KUKA KRL program: ho_com_02_ag01_g01.src, ho_com_02_ag01_g01.dat

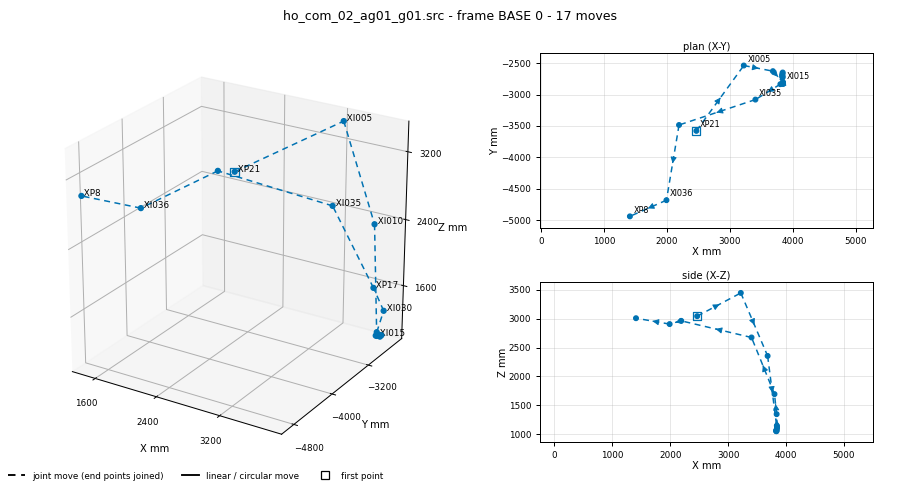
[picture p0: tool path of ho_com_02_ag01_g01.src in frame BASE 0, 17 of 17 moves have a stored position in this frame; points joined in program order, loops and branches not executed]
--- ho_com_02_ag01_g01.src ---
&ACCESS RVO4
&REL 568
&COMMENT Pega Traseira LTA-LTB
&PARAM DISKPATH = KRC:\R1\Program\MANIPULACAO NTC
DEF HO_COM_02_AG01_G01 ( )
;FOLD INI
  ;FOLD BASISTECH INI
    GLOBAL INTERRUPT DECL 3 WHEN $STOPMESS==TRUE DO IR_STOPM ( )
    INTERRUPT ON 3
    BAS (#INITMOV,0)
  ;ENDFOLD (BASISTECH INI)
;FOLD GRIPPERTECH INI
USER_GRP(0,DUMMY,DUMMY,GDEFAULT)
;ENDFOLD (GRIPPERTECH INI)
  ;FOLD USER INI
    ;Make your modifications here

  ;ENDFOLD (USER INI)
;ENDFOLD (INI)

; Caracterizacao dos meios de producao
; Changes: Pega Traseira no AGV
; Modelos: Axor/Atego - LTA/LTB
; Versao Atual: 05/01/2016
; Ferramenta: Gripper 903
; Name: P13.050-R1

chk_w9_wechs_ok ( ) ;CHECK GRIPPER 903

;FOLD PTP P21 CONT Vel=100 % PDAT15 Tool[10]:Grp 903 c/ pc Base[0];%{PE}%R 8.2.20,%MKUKATPBASIS,%CMOVE,%VPTP,%P 1:PTP, 2:P21, 3:C_DIS, 5:100, 7:PDAT15
$BWDSTART=FALSE
PDAT_ACT=PPDAT15
FDAT_ACT=FP21
BAS(#PTP_PARAMS,100)
PTP XP21 C_DIS
;ENDFOLD

;FOLD WAIT FOR ( NOT IN 581 'DK 8 GRP Axor 903 Tampa R' ) AND ( IN 582 'DK 8 GRP Axor 903 Tampa V' );%{PE}%R 8.2.20,%MKUKATPBASIS,%CEXT_WAIT_FOR,%VEXT_WAIT_FOR,%P 2:, 4:NOT, 5:$IN, 6:581, 7:DK 8 GRP Axor 903 Tampa R, 9:AND, 10:, 12:, 13:$IN, 14:582, 15:DK 8 GRP Axor 903 Tampa V, 17:
WAIT FOR  (  NOT $IN[581] ) AND ( $IN[582] )
;ENDFOLD
;FOLD WAIT FOR ( NOT IN 489 'Presença de peça 1 - Axor 903' ) AND ( NOT IN 490 'Presença de peça 2 - Axor 903' );%{PE}%R 8.2.20,%MKUKATPBASIS,%CEXT_WAIT_FOR,%VEXT_WAIT_FOR,%P 2:, 4:NOT, 5:$IN, 6:489, 7:Presença de peça 1 - Axor 903, 9:AND, 10:, 12:NOT, 13:$IN, 14:490, 15:Presença de peça 2 - Axor 903, 17:
WAIT FOR  (  NOT $IN[489] ) AND (  NOT $IN[490] )
;ENDFOLD

; ABRE GRAMPOS
;FOLD SET Z1.1/2 GRP AXOR 903 State=OPN CONT at START Delay=1 ms;%{PE}%R 8.2.1,%MKUKATPGRP,%CGRP,%VGRP,%P 2:7, 4:1, 5:#YES, 6:GDAT19, 8:0, 10:1
TRIGGER WHEN DISTANCE=0 DELAY=1 DO H50(GRP_APO,7,1,GCONT) PRIO=-1
;ENDFOLD
;FOLD SET Z2.1/2 RPS AXOR 903 State=OPN CONT at START Delay=1 ms;%{PE}%R 8.2.1,%MKUKATPGRP,%CGRP,%VGRP,%P 2:8, 4:1, 5:#YES, 6:GDAT23, 8:0, 10:1
TRIGGER WHEN DISTANCE=0 DELAY=1 DO H50(GRP_APO,8,1,GCONT) PRIO=-1
;ENDFOLD
;FOLD SET Z3.1 GRP AXOR 903 State=OPN CONT at START Delay=1 ms;%{PE}%R 8.2.1,%MKUKATPGRP,%CGRP,%VGRP,%P 2:9, 4:1, 5:#YES, 6:GDAT21, 8:0, 10:1
TRIGGER WHEN DISTANCE=0 DELAY=1 DO H50(GRP_APO,9,1,GCONT) PRIO=-1
;ENDFOLD
;FOLD SET Z7.1 GRP 7 AXOR 903 State=OPN CONT at START Delay=1 ms;%{PE}%R 8.2.1,%MKUKATPGRP,%CGRP,%VGRP,%P 2:14, 4:1, 5:#YES, 6:GDAT27, 8:0, 10:1
TRIGGER WHEN DISTANCE=0 DELAY=1 DO H50(GRP_APO,14,1,GCONT) PRIO=-1
;ENDFOLD
;FOLD SET Z6.1 VAC AXOR 903 State=CONT at START Delay=1 ms;%{PE}%R 8.2.1,%MKUKATPGRP,%CGRP,%VGRP,%P 2:13, 4:2, 5:#YES, 6:GDAT28, 8:0, 10:1
TRIGGER WHEN DISTANCE=0 DELAY=1 DO H50(GRP_APO,13,2,GCONT) PRIO=-1
;ENDFOLD
;FOLD SET Z6.1 VAC AXOR 903 State=OFF CONT at START Delay=1 ms;%{PE}%R 8.2.1,%MKUKATPGRP,%CGRP,%VGRP,%P 2:13, 4:3, 5:#YES, 6:GDAT29, 8:0, 10:1
TRIGGER WHEN DISTANCE=0 DELAY=1 DO H50(GRP_APO,13,3,GCONT) PRIO=-1
;ENDFOLD
chk_w9_grp1_opn( )
chk_w9_rps2_opn( )
chk_w9_grp3_opn( )
chk_w9_grp4_opn( )
chk_w9_grp5_vac_off( )

;AGUARDA LIBERACAO DE PEGA
;FOLD OUT 3370 'Lib. p/ Pegar Parede Traseira' State=TRUE ;%{PE}%R 8.2.20,%MKUKATPBASIS,%COUT,%VOUTX,%P 2:3370, 3:Lib. p/ Pegar Parede Traseira, 5:TRUE, 6:
$OUT[3370]=TRUE
;ENDFOLD
;FOLD WAIT FOR ( IN 3370 'Aguarda Lib. p/ Retirar Parede Traseira' );%{PE}%R 8.2.20,%MKUKATPBASIS,%CEXT_WAIT_FOR,%VEXT_WAIT_FOR,%P 2:, 4:, 5:$IN, 6:3370, 7:Aguarda Lib. p/ Retirar Parede Traseira, 9:
WAIT FOR  ( $IN[3370] )
;ENDFOLD
;FOLD OUT 3370 'Lib. p/ Pegar Parede Traseira' State=FALSE ;%{PE}%R 8.2.20,%MKUKATPBASIS,%COUT,%VOUTX,%P 2:3370, 3:Lib. p/ Pegar Parede Traseira, 5:FALSE, 6:
$OUT[3370]=FALSE
;ENDFOLD
;FOLD OUT 3342 'Fora area externa' State=FALSE ;%{PE}%R 8.2.20,%MKUKATPBASIS,%COUT,%VOUTX,%P 2:3342, 3:Fora area externa, 5:FALSE, 6:
$OUT[3342]=FALSE
;ENDFOLD

;FOLD PTP l005 CONT Vel=100 % P_OLP2 Tool[10]:Grp 903 c/ pc Base[0];%{PE}%R 8.2.20,%MKUKATPBASIS,%CMOVE,%VPTP,%P 1:PTP, 2:l005, 3:C_DIS, 5:100, 7:P_OLP2
$BWDSTART=FALSE
PDAT_ACT=PP_OLP2
FDAT_ACT=Fl005
BAS(#PTP_PARAMS,100)
PTP Xl005 C_DIS
;ENDFOLD
;FOLD PTP l010 CONT Vel=100 % P_OLP3 Tool[10]:Grp 903 c/ pc Base[0];%{PE}%R 8.2.20,%MKUKATPBASIS,%CMOVE,%VPTP,%P 1:PTP, 2:l010, 3:C_DIS, 5:100, 7:P_OLP3
$BWDSTART=FALSE
PDAT_ACT=PP_OLP3
FDAT_ACT=Fl010
BAS(#PTP_PARAMS,100)
PTP Xl010 C_DIS
;ENDFOLD
;FOLD PTP l015 CONT Vel=100 % P_OLP4 Tool[10]:Grp 903 c/ pc Base[0];%{PE}%R 8.2.20,%MKUKATPBASIS,%CMOVE,%VPTP,%P 1:PTP, 2:l015, 3:C_DIS, 5:100, 7:P_OLP4
$BWDSTART=FALSE
PDAT_ACT=PP_OLP4
FDAT_ACT=Fl015
BAS(#PTP_PARAMS,100)
PTP Xl015 C_DIS
;ENDFOLD
;FOLD LIN P15 CONT Vel=2 m/s CPDAT3 Tool[10]:Grp 903 c/ pc Base[0];%{PE}%R 8.2.20,%MKUKATPBASIS,%CMOVE,%VLIN,%P 1:LIN, 2:P15, 3:C_DIS C_DIS, 5:2, 7:CPDAT3
$BWDSTART=FALSE
LDAT_ACT=LCPDAT3
FDAT_ACT=FP15
BAS(#CP_PARAMS,2)
LIN XP15 C_DIS C_DIS
;ENDFOLD
;FOLD LIN P9 CONT Vel=1 m/s CPDAT1 Tool[10]:Grp 903 c/ pc Base[0];%{PE}%R 8.2.20,%MKUKATPBASIS,%CMOVE,%VLIN,%P 1:LIN, 2:P9, 3:C_DIS C_DIS, 5:1, 7:CPDAT1
$BWDSTART=FALSE
LDAT_ACT=LCPDAT1
FDAT_ACT=FP9
BAS(#CP_PARAMS,1)
LIN XP9 C_DIS C_DIS
;ENDFOLD

; POSICAO DE PEGA AXOR/ATEGO LTA-LTB
;FOLD LIN P_PE02 Vel=0.25 m/s CPDAT4 Tool[9]:Grp 903 s/ pc Base[0];%{PE}%R 8.2.20,%MKUKATPBASIS,%CMOVE,%VLIN,%P 1:LIN, 2:P_PE02, 3:, 5:0.25, 7:CPDAT4
$BWDSTART=FALSE
LDAT_ACT=LCPDAT4
FDAT_ACT=FP_PE02
BAS(#CP_PARAMS,0.25)
LIN XP_PE02
;ENDFOLD

IF (NOT(GHOST())) THEN
;FOLD WAIT FOR ( IN 489 'Presença de peça 1 - Axor 903' ) AND ( IN 490 'Presença de peça 2 - Axor 903' );%{PE}%R 8.2.20,%MKUKATPBASIS,%CEXT_WAIT_FOR,%VEXT_WAIT_FOR,%P 2:, 4:, 5:$IN, 6:489, 7:Presença de peça 1 - Axor 903, 9:AND, 10:, 12:, 13:$IN, 14:490, 15:Presença de peça 2 - Axor 903, 17:
WAIT FOR  ( $IN[489] ) AND ( $IN[490] )
;ENDFOLD
ENDIF

; FECHA GRAMPOS
;FOLD SET Z2.1/2 RPS AXOR 903 State=CLO GDAT22;%{PE}%R 8.2.1,%MKUKATPGRP,%CGRP,%VGRP,%P 2:8, 4:2, 5:#NO, 6:GDAT22, 8:0, 10:0
H50(GRP,8,2,GGDAT22)
;ENDFOLD
;FOLD SET Z1.1/2 GRP AXOR 903 State=CLO GDAT16;%{PE}%R 8.2.1,%MKUKATPGRP,%CGRP,%VGRP,%P 2:7, 4:2, 5:#NO, 6:GDAT16, 8:0, 10:0
H50(GRP,7,2,GGDAT16)
;ENDFOLD
;FOLD SET Z3.1 GRP AXOR 903 State=CLO GDAT18;%{PE}%R 8.2.1,%MKUKATPGRP,%CGRP,%VGRP,%P 2:9, 4:2, 5:#NO, 6:GDAT18, 8:0, 10:0
H50(GRP,9,2,GGDAT18)
;ENDFOLD
;FOLD SET Z7.1 GRP 7 AXOR 903 State=CLO GDAT32;%{PE}%R 8.2.1,%MKUKATPGRP,%CGRP,%VGRP,%P 2:14, 4:2, 5:#NO, 6:GDAT32, 8:0, 10:0
H50(GRP,14,2,GGDAT32)
;ENDFOLD
chk_w9_rps2_clo( )
chk_w9_grp1_clo( )
chk_w9_grp3_clo( )
chk_w9_grp4_clo( )

IF (NOT(GHOST())) THEN
;FOLD SET Z6.1 VAC AXOR 903 State=VACUUM GDAT31;%{PE}%R 8.2.1,%MKUKATPGRP,%CGRP,%VGRP,%P 2:13, 4:1, 5:#NO, 6:GDAT31, 8:0, 10:0
H50(GRP,13,1,GGDAT31)
;ENDFOLD
chk_w9_grp5_vac_on( )
ENDIF

;AGUARDA LIBERACAO SAIR COM PECA
;FOLD OUT 3371 'Lib. p/ Sair c/ Parede Traseira' State=TRUE ;%{PE}%R 8.2.20,%MKUKATPBASIS,%COUT,%VOUTX,%P 2:3371, 3:Lib. p/ Sair c/ Parede Traseira, 5:TRUE, 6:
$OUT[3371]=TRUE
;ENDFOLD
;FOLD WAIT FOR ( IN 3371 'Aguarda Lib. p/ Sair c/ Parede Traseira' );%{PE}%R 8.2.20,%MKUKATPBASIS,%CEXT_WAIT_FOR,%VEXT_WAIT_FOR,%P 2:, 4:, 5:$IN, 6:3371, 7:Aguarda Lib. p/ Sair c/ Parede Traseira, 9:
WAIT FOR  ( $IN[3371] )
;ENDFOLD
;FOLD OUT 3371 'Lib. p/ Sair c/ Parede Traseira' State=FALSE ;%{PE}%R 8.2.20,%MKUKATPBASIS,%COUT,%VOUTX,%P 2:3371, 3:Lib. p/ Sair c/ Parede Traseira, 5:FALSE, 6:
$OUT[3371]=FALSE
;ENDFOLD
;FOLD WAIT FOR ( IN 582 'DK 8 GRP Axor 903 Tampa V' );%{PE}%R 8.2.20,%MKUKATPBASIS,%CEXT_WAIT_FOR,%VEXT_WAIT_FOR,%P 2:, 4:, 5:$IN, 6:582, 7:DK 8 GRP Axor 903 Tampa V, 9:
WAIT FOR  ( $IN[582] )
;ENDFOLD

;FOLD LIN P11 Vel=0.25 m/s CPDAT2 Tool[10]:Grp 903 c/ pc Base[0];%{PE}%R 8.2.20,%MKUKATPBASIS,%CMOVE,%VLIN,%P 1:LIN, 2:P11, 3:, 5:0.25, 7:CPDAT2
$BWDSTART=FALSE
LDAT_ACT=LCPDAT2
FDAT_ACT=FP11
BAS(#CP_PARAMS,0.25)
LIN XP11
;ENDFOLD

IF (NOT(GHOST())) THEN
;FOLD WAIT FOR ( IN 489 'Presença de peça 1 - Axor 903' ) AND ( IN 490 'Presença de peça 2 - Axor 903' );%{PE}%R 8.2.20,%MKUKATPBASIS,%CEXT_WAIT_FOR,%VEXT_WAIT_FOR,%P 2:, 4:, 5:$IN, 6:489, 7:Presença de peça 1 - Axor 903, 9:AND, 10:, 12:, 13:$IN, 14:490, 15:Presença de peça 2 - Axor 903, 17:
WAIT FOR  ( $IN[489] ) AND ( $IN[490] )
;ENDFOLD
ENDIF

;FOLD LIN l020 CONT Vel=0.4 m/s L_OLP2 Tool[10]:Grp 903 c/ pc Base[0];%{PE}%R 8.2.20,%MKUKATPBASIS,%CMOVE,%VLIN,%P 1:LIN, 2:l020, 3:C_DIS C_DIS, 5:0.4, 7:L_OLP2
$BWDSTART=FALSE
LDAT_ACT=LL_OLP2
FDAT_ACT=Fl020
BAS(#CP_PARAMS,0.4)
LIN Xl020 C_DIS C_DIS
;ENDFOLD
;FOLD PTP P10 CONT Vel=100 % PDAT5 Tool[10]:Grp 903 c/ pc Base[0];%{PE}%R 8.2.20,%MKUKATPBASIS,%CMOVE,%VPTP,%P 1:PTP, 2:P10, 3:C_DIS, 5:100, 7:PDAT5
$BWDSTART=FALSE
PDAT_ACT=PPDAT5
FDAT_ACT=FP10
BAS(#PTP_PARAMS,100)
PTP XP10 C_DIS
;ENDFOLD
;FOLD PTP P12 CONT Vel=100 % PDAT6 Tool[10]:Grp 903 c/ pc Base[0];%{PE}%R 8.2.20,%MKUKATPBASIS,%CMOVE,%VPTP,%P 1:PTP, 2:P12, 3:C_DIS, 5:100, 7:PDAT6
$BWDSTART=FALSE
PDAT_ACT=PPDAT6
FDAT_ACT=FP12
BAS(#PTP_PARAMS,100)
PTP XP12 C_DIS
;ENDFOLD
;FOLD PTP l030 CONT Vel=50 % P_OLP6 Tool[10]:Grp 903 c/ pc Base[0];%{PE}%R 8.2.20,%MKUKATPBASIS,%CMOVE,%VPTP,%P 1:PTP, 2:l030, 3:C_DIS, 5:50, 7:P_OLP6
$BWDSTART=FALSE
PDAT_ACT=PP_OLP6
FDAT_ACT=Fl030
BAS(#PTP_PARAMS,50)
PTP Xl030 C_DIS
;ENDFOLD
;FOLD PTP P17 CONT Vel=50 % PDAT10 Tool[10]:Grp 903 c/ pc Base[0];%{PE}%R 8.2.20,%MKUKATPBASIS,%CMOVE,%VPTP,%P 1:PTP, 2:P17, 3:C_DIS, 5:50, 7:PDAT10
$BWDSTART=FALSE
PDAT_ACT=PPDAT10
FDAT_ACT=FP17
BAS(#PTP_PARAMS,50)
PTP XP17 C_DIS
;ENDFOLD
;FOLD PTP l035 CONT Vel=50 % P_OLP7 Tool[10]:Grp 903 c/ pc Base[0];%{PE}%R 8.2.20,%MKUKATPBASIS,%CMOVE,%VPTP,%P 1:PTP, 2:l035, 3:C_DIS, 5:50, 7:P_OLP7
$BWDSTART=FALSE
PDAT_ACT=PP_OLP7
FDAT_ACT=Fl035
BAS(#PTP_PARAMS,50)
PTP Xl035 C_DIS
;ENDFOLD
;FOLD PTP P18 CONT Vel=30 % PDAT11 Tool[10]:Grp 903 c/ pc Base[0];%{PE}%R 8.2.20,%MKUKATPBASIS,%CMOVE,%VPTP,%P 1:PTP, 2:P18, 3:C_DIS, 5:30, 7:PDAT11
$BWDSTART=FALSE
PDAT_ACT=PPDAT11
FDAT_ACT=FP18
BAS(#PTP_PARAMS,30)
PTP XP18 C_DIS
;ENDFOLD
;FOLD PTP l036 CONT Vel=30 % P_OLP9 Tool[10]:Grp 903 c/ pc Base[0];%{PE}%R 8.2.20,%MKUKATPBASIS,%CMOVE,%VPTP,%P 1:PTP, 2:l036, 3:C_DIS, 5:30, 7:P_OLP9
$BWDSTART=FALSE
PDAT_ACT=PP_OLP9
FDAT_ACT=Fl036
BAS(#PTP_PARAMS,30)
PTP Xl036 C_DIS
;ENDFOLD

;LIBERA AREA
;FOLD PULSE 3349 'R1 pegou peça' State=TRUE Time=3 sec;%{PE}%R 8.2.20,%MKUKATPBASIS,%COUT,%VPULSE,%P 2:3349, 3:R1 pegou peça, 5:TRUE, 6:, 8:3
PULSE($OUT[3349], TRUE,3)
;ENDFOLD
;FOLD OUT 3342 'Fora area externa' State=TRUE ;%{PE}%R 8.2.20,%MKUKATPBASIS,%COUT,%VOUTX,%P 2:3342, 3:Fora area externa, 5:TRUE, 6:
$OUT[3342]=TRUE
;ENDFOLD

;FOLD PTP P8 CONT Vel=30 % PDAT4 Tool[10]:Grp 903 c/ pc Base[0];%{PE}%R 8.2.20,%MKUKATPBASIS,%CMOVE,%VPTP,%P 1:PTP, 2:P8, 3:C_DIS, 5:30, 7:PDAT4
$BWDSTART=FALSE
PDAT_ACT=PPDAT4
FDAT_ACT=FP8
BAS(#PTP_PARAMS,30)
PTP XP8 C_DIS
;ENDFOLD

END

--- ho_com_02_ag01_g01.dat ---
&ACCESS RVO4
&REL 568
&COMMENT Pega Traseira LTA-LTB
&PARAM DISKPATH = KRC:\R1\Program\MANIPULACAO NTC
DEFDAT  ho_com_02_ag01_g01
;FOLD EXTERNAL DECLARATIONS;%{PE}%MKUKATPBASIS,%CEXT,%VCOMMON,%P
;FOLD GRIPPERTECH EXT
EXT  H50 (INT  :IN,INT  :IN,INT  :IN,GRP_TYP  :IN )
;ENDFOLD (GRIPPERTECH EXT)
;FOLD SPOTTECH EXT
EXT  USERSPOT (S_COMMAND  :IN,SPOT_TYPE  :IN )
;ENDFOLD (SPOTTECH EXT)
;FOLD BASISTECH EXT;%{PE}%MKUKATPBASIS,%CEXT,%VEXT,%P
EXT  BAS (BAS_COMMAND  :IN,REAL  :IN )
DECL INT SUCCESS
;ENDFOLD (BASISTECH EXT)
;FOLD USER EXT;%{E}%MKUKATPUSER,%CEXT,%VEXT,%P
;Make your modifications here

;ENDFOLD (USER EXT)
DECL FDAT Fl005={TOOL_NO 9,BASE_NO 0,IPO_FRAME #BASE,POINT2[] " ",TQ_STATE FALSE}
DECL PDAT PP_OLP2={VEL 100.0,ACC 100.0,APO_DIST 10.0,APO_MODE #CDIS}
DECL E6POS Xl005={X 3218.60791,Y -2539.229,Z 3442.36011,A -30.2562904,B 46.8825684,C -113.404999,S 2,T 11,E1 -3250.0,E2 0.0,E3 0.0,E4 0.0,E5 0.0,E6 0.0}
DECL FDAT Fl010={TOOL_NO 9,BASE_NO 0,IPO_FRAME #BASE,POINT2[] " "}
DECL PDAT PP_OLP3={VEL 100.0,ACC 100.0,APO_DIST 10.0,APO_MODE #CDIS}
DECL E6POS Xl010={X 3681.40308,Y -2628.80493,Z 2354.81299,A -52.0649681,B 58.5603714,C -139.654205,S 2,T 11,E1 -3426.1709,E2 0.0,E3 0.0,E4 0.0,E5 0.0,E6 0.0}
DECL FDAT Fl015={TOOL_NO 9,BASE_NO 0,IPO_FRAME #BASE,POINT2[] " "}
DECL PDAT PP_OLP4={VEL 100.0,ACC 100.0,APO_DIST 10.0,APO_MODE #CDIS}
DECL E6POS Xl015={X 3842.71606,Y -2807.72095,Z 1105.85901,A -89.6218338,B 67.1568527,C 178.501907,S 2,T 11,E1 -3522.73389,E2 0.0,E3 0.0,E4 0.0,E5 0.0,E6 0.0}
DECL FDAT FP_PE02={TOOL_NO 9,BASE_NO 0,IPO_FRAME #BASE,POINT2[] " ",TQ_STATE FALSE}
DECL E6POS XP_PE02={X 3830.49609,Y -2675.78906,Z 1055.40906,A -88.9839935,B 65.9510117,C 179.429596,S 2,T 11,E1 -3701.05493,E2 0.0,E3 0.0,E4 0.0,E5 0.0,E6 0.0}
DECL FDAT Fl020={TOOL_NO 10,BASE_NO 0,IPO_FRAME #BASE,POINT2[] " "}
DECL E6POS Xl020={X 3835.47607,Y -2731.25488,Z 1079.94604,A -89.6218033,B 67.1567001,C 178.501999,S 2,T 11,E1 -3700.23511,E2 0.0,E3 0.0,E4 0.0,E5 0.0,E6 0.0}
DECL LDAT LL_OLP2={VEL 0.25,ACC 100.0,APO_DIST 30.0,APO_FAC 0.0,ORI_TYP #VAR,CIRC_TYP #BASE,JERK_FAC 50.0}
DECL FDAT Fl030={TOOL_NO 10,BASE_NO 0,IPO_FRAME #BASE,POINT2[] " "}
DECL PDAT PP_OLP6={VEL 100.0,ACC 70.0,APO_DIST 50.0,APO_MODE #CDIS}
DECL E6POS Xl030={X 3837.04712,Y -2650.14209,Z 1349.71301,A 0.0,B 89.9999466,C -92.2000885,S 2,T 11,E1 -3700.00098,E2 0.0,E3 0.0,E4 0.0,E5 0.0,E6 0.0}
DECL FDAT Fl035={TOOL_NO 10,BASE_NO 0,IPO_FRAME #BASE,POINT2[] " ",TQ_STATE FALSE}
DECL PDAT PP_OLP7={VEL 100.0,ACC 50.0,APO_DIST 50.0,APO_MODE #CDIS}
DECL E6POS Xl035={X 3403.61108,Y -3080.45508,Z 2673.61792,A 76.7603836,B 73.9680481,C -4.25617409,S 2,T 11,E1 -3973.10107,E2 0.0,E3 0.0,E4 0.0,E5 0.0,E6 0.0}
DECL BASIS_SUGG_T LAST_BASIS={POINT1[] "P22                     ",POINT2[] "P22                     ",CP_PARAMS[] "CPDAT3                  ",PTP_PARAMS[] "PDAT16                  ",CONT[] "                        ",CP_VEL[] "0.4                     ",PTP_VEL[] "100                     ",SYNC_PARAMS[] "SYNCDAT                 ",SPL_NAME[] "S0                      "}
DECL PDAT PP_OLP9={VEL 100.0,ACC 50.0,APO_DIST 50.0,APO_MODE #CDIS}
DECL E6POS Xl036={X 1989.90601,Y -4679.04883,Z 2904.58691,A -29.6459503,B 80.8687363,C -48.2684593,S 2,T 11,E1 -3220.72095,E2 0.0,E3 0.0,E4 0.0,E5 0.0,E6 0.0}
DECL FDAT Fl036={TOOL_NO 10,BASE_NO 0,IPO_FRAME #BASE,POINT2[] " ",TQ_STATE FALSE}
DECL GRP_SUGG_T LAST_GRP={NUMBER[] "13                      ",STATE[] "3                       ",PARAMS[] "GDAT29                  "}
DECL GRP_TYP GGDAT4={G_APO #NO,GRP_TIME 0.200000003,CTRL #OFF,DLY 0,DST 1}
DECL GRP_TYP GGDAT6={G_APO #NO,GRP_TIME 0.200000003,CTRL #OFF,DLY 0,DST 1}
DECL GRP_TYP GGDAT8={G_APO #NO,GRP_TIME 0.200000003,CTRL #OFF,DLY 0,DST 1}
DECL GRP_TYP GGDAT5={G_APO #NO,GRP_TIME 0.200000003,CTRL #OFF,DLY 0,DST 1}
DECL GRP_TYP GGDAT7={G_APO #NO,GRP_TIME 0.200000003,CTRL #OFF,DLY 0,DST 1}
DECL GRP_TYP GGDAT9={G_APO #NO,GRP_TIME 0.200000003,CTRL #OFF,DLY 0,DST 1}
DECL GRP_TYP GGDAT10={G_APO #NO,GRP_TIME 0.200000003,CTRL #OFF,DLY 0,DST 1}
DECL GRP_TYP GGDAT11={G_APO #NO,GRP_TIME 0.200000003,CTRL #OFF,DLY 0,DST 1}
DECL GRP_TYP GGDAT12={G_APO #NO,GRP_TIME 0.200000003,CTRL #OFF,DLY 0,DST 1}
DECL GRP_TYP GGDAT13={G_APO #NO,GRP_TIME 0.200000003,CTRL #OFF,DLY 0,DST 1}
DECL GRP_TYP GGDAT14={G_APO #NO,GRP_TIME 0.200000003,CTRL #OFF,DLY 0,DST 1}
DECL GRP_TYP GGDAT15={G_APO #NO,GRP_TIME 0.200000003,CTRL #OFF,DLY 0,DST 1}
DECL GRP_TYP GGDAT16={G_APO #NO,GRP_TIME 0.200000003,CTRL #OFF,DLY 0,DST 1}
DECL GRP_TYP GGDAT17={G_APO #NO,GRP_TIME 0.200000003,CTRL #OFF,DLY 0,DST 1}
DECL GRP_TYP GGDAT18={G_APO #NO,GRP_TIME 0.200000003,CTRL #OFF,DLY 0,DST 1}
DECL E6POS XP8={X 1408.87598,Y -4935.90723,Z 3006.11108,A -20.0040207,B 69.0891495,C -21.5691395,S 2,T 11,E1 -3220.81396,E2 0.0,E3 0.0,E4 0.0,E5 0.0,E6 0.0}
DECL FDAT FP8={TOOL_NO 10,BASE_NO 0,IPO_FRAME #BASE,POINT2[] " ",TQ_STATE FALSE}
DECL PDAT PPDAT4={VEL 100.0,ACC 50.0,APO_DIST 50.0,APO_MODE #CDIS}
DECL GRP_TYP GGDAT19={G_APO #NO,GRP_TIME 0.200000003,CTRL #OFF,DLY 0,DST 1}
DECL GRP_TYP GGDAT20={G_APO #NO,GRP_TIME 0.200000003,CTRL #OFF,DLY 0,DST 1}
DECL GRP_TYP GGDAT21={G_APO #NO,GRP_TIME 0.200000003,CTRL #OFF,DLY 0,DST 1}
DECL E6POS XP9={X 3831.39795,Y -2694.11499,Z 1062.47095,A -89.3210831,B 67.2410583,C 178.401596,S 2,T 11,E1 -3706.729,E2 0.0,E3 0.0,E4 0.0,E5 0.0,E6 0.0}
DECL FDAT FP9={TOOL_NO 9,BASE_NO 0,IPO_FRAME #BASE,POINT2[] " ",TQ_STATE FALSE}
DECL LDAT LCPDAT1={VEL 2.0,ACC 100.0,APO_DIST 50.0,APO_FAC 50.0,AXIS_VEL 100.0,AXIS_ACC 100.0,ORI_TYP #VAR,CIRC_TYP #BASE,JERK_FAC 50.0,GEAR_JERK 50.0,EXAX_IGN 0}
DECL E6POS XP10={X 3843.63696,Y -2833.05688,Z 1120.75305,A -90.5353394,B 75.7654572,C 177.633301,S 2,T 11,E1 -3700.06592,E2 0.0,E3 0.0,E4 0.0,E5 0.0,E6 0.0}
DECL FDAT FP10={TOOL_NO 10,BASE_NO 0,IPO_FRAME #BASE,POINT2[] " ",TQ_STATE FALSE}
DECL PDAT PPDAT5={VEL 100.0,ACC 100.0,APO_DIST 30.0,APO_MODE #CDIS}
DECL E6POS XP11={X 3832.33203,Y -2715.6731,Z 1068.93896,A -89.3303986,B 65.348587,C 178.376099,S 2,T 11,E1 -3700.04199,E2 0.0,E3 0.0,E4 0.0,E5 0.0,E6 0.0}
DECL FDAT FP11={TOOL_NO 10,BASE_NO 0,IPO_FRAME #BASE,POINT2[] " ",TQ_STATE FALSE}
DECL LDAT LCPDAT2={VEL 2.0,ACC 100.0,APO_DIST 5.0,APO_FAC 50.0,AXIS_VEL 100.0,AXIS_ACC 100.0,ORI_TYP #VAR,CIRC_TYP #BASE,JERK_FAC 50.0,GEAR_JERK 50.0,EXAX_IGN 0}
DECL E6POS XP12={X 3840.92993,Y -2806.29492,Z 1150.78198,A -88.0371933,B 77.8013535,C -179.918396,S 2,T 11,E1 -3700.88989,E2 0.0,E3 0.0,E4 0.0,E5 0.0,E6 0.0}
DECL FDAT FP12={TOOL_NO 10,BASE_NO 0,IPO_FRAME #BASE,POINT2[] " ",TQ_STATE FALSE}
DECL PDAT PPDAT6={VEL 100.0,ACC 100.0,APO_DIST 30.0,APO_MODE #CDIS}
DECL LDAT LCPDAT3={VEL 2.0,ACC 100.0,APO_DIST 50.0,APO_FAC 50.0,AXIS_VEL 100.0,AXIS_ACC 100.0,ORI_TYP #VAR,CIRC_TYP #BASE,JERK_FAC 50.0,GEAR_JERK 50.0,EXAX_IGN 0}
DECL E6POS XP15={X 3833.42603,Y -2714.77393,Z 1055.72803,A -89.0524368,B 67.2397308,C 178.692993,S 2,T 11,E1 -3703.71997,E2 0.0,E3 0.0,E4 0.0,E5 0.0,E6 0.0}
DECL FDAT FP15={TOOL_NO 9,BASE_NO 0,IPO_FRAME #BASE,POINT2[] " ",TQ_STATE FALSE}
DECL GRP_TYP GGDAT22={G_APO #NO,GRP_TIME 0.200000003,CTRL #OFF,DLY 0,DST 1}
DECL GRP_TYP GGDAT23={G_APO #NO,GRP_TIME 0.200000003,CTRL #OFF,DLY 0,DST 1}
DECL GRP_TYP GGDAT3={G_APO #NO,GRP_TIME 0.200000003,CTRL #OFF,DLY 0,DST 1}
DECL GRP_TYP GGDAT1={G_APO #NO,GRP_TIME 0.200000003,CTRL #OFF,DLY 0,DST 1}
DECL GRP_TYP GGDAT2={G_APO #NO,GRP_TIME 0.200000003,CTRL #OFF,DLY 0,DST 1}
DECL GRP_TYP GGDAT24={G_APO #NO,GRP_TIME 0.200000003,CTRL #OFF,DLY 0,DST 1}
DECL E6POS XP17={X 3800.02808,Y -2835.55811,Z 1695.61401,A 77.3357925,B 87.3917465,C -11.0309896,S 2,T 11,E1 -3820.08398,E2 0.0,E3 0.0,E4 0.0,E5 0.0,E6 0.0}
DECL FDAT FP17={TOOL_NO 10,BASE_NO 0,IPO_FRAME #BASE,POINT2[] " ",TQ_STATE FALSE}
DECL PDAT PPDAT10={VEL 100.0,ACC 50.0,APO_DIST 50.0,APO_MODE #CDIS}
DECL E6POS XP18={X 2189.81909,Y -3484.28491,Z 2960.64111,A -23.6490192,B 79.1503906,C -53.971241,S 2,T 11,E1 -2223.51489,E2 0.0,E3 0.0,E4 0.0,E5 0.0,E6 0.0}
DECL FDAT FP18={TOOL_NO 10,BASE_NO 0,IPO_FRAME #BASE,POINT2[] " ",TQ_STATE FALSE}
DECL PDAT PPDAT11={VEL 100.0,ACC 50.0,APO_DIST 50.0,APO_MODE #CDIS}
DECL LDAT LCPDAT4={VEL 2.0,ACC 100.0,APO_DIST 100.0,APO_FAC 50.0,AXIS_VEL 100.0,AXIS_ACC 100.0,ORI_TYP #VAR,CIRC_TYP #BASE,JERK_FAC 50.0,GEAR_JERK 50.0,EXAX_IGN 0}
DECL GRP_TYP GGDAT25={G_APO #NO,GRP_TIME 0.200000003,CTRL #OFF,DLY 0,DST 1}
DECL GRP_TYP GGDAT26={G_APO #NO,GRP_TIME 0.200000003,CTRL #OFF,DLY 0,DST 1}
DECL GRP_TYP GGDAT27={G_APO #NO,GRP_TIME 0.200000003,CTRL #OFF,DLY 0,DST 1}
DECL GRP_TYP GGDAT28={G_APO #NO,GRP_TIME 0.200000003,CTRL #OFF,DLY 0,DST 1}
DECL GRP_TYP GGDAT29={G_APO #NO,GRP_TIME 0.200000003,CTRL #OFF,DLY 0,DST 1}
DECL GRP_TYP GGDAT30={G_APO #NO,GRP_TIME 0.200000003,CTRL #OFF,DLY 0,DST 1}
DECL GRP_TYP GGDAT31={G_APO #NO,GRP_TIME 0.200000003,CTRL #OFF,DLY 0,DST 1}
DECL GRP_TYP GGDAT32={G_APO #NO,GRP_TIME 0.200000003,CTRL #OFF,DLY 0,DST 1}
DECL GRP_TYP GCONT={G_APO #YES,GRP_TIME 0.0,CTRL #OFF,DLY 0,DST 0}
DECL PDAT PPDAT15={VEL 100.0,ACC 100.0,APO_DIST 50.0,APO_MODE #CDIS}
DECL E6POS XP21={X 2465.09399,Y -3577.50903,Z 3041.33594,A -31.7606792,B 68.6130829,C -82.8799362,S 2,T 11,E1 -3229.75,E2 0.0,E3 0.0,E4 0.0,E5 0.0,E6 0.0}
DECL FDAT FP21={TOOL_NO 9,BASE_NO 0,IPO_FRAME #BASE,POINT2[] " ",TQ_STATE FALSE}
DECL E6POS XP22={X 1678.52698,Y -2966.29492,Z 1407.29797,A -178.796707,B -1.65615797,C 178.619003,S 2,T 3,E1 -1997.12695,E2 0.0,E3 0.0,E4 0.0,E5 0.0,E6 0.0}
DECL FDAT FP22={TOOL_NO 9,BASE_NO 0,IPO_FRAME #BASE,POINT2[] " ",TQ_STATE FALSE}
DECL PDAT PPDAT16={VEL 100.0,ACC 100.0,APO_DIST 100.0,APO_MODE #CDIS}
ENDDAT
